FUNCTION_BLOCK Doors (* Composite Function Block Type *)
  (* Standard: 61499-2 *)
  (* Version 0.0, 11/8/2016, Dmitry, nxtControl GmbH, template *)
  PACKAGE Main;
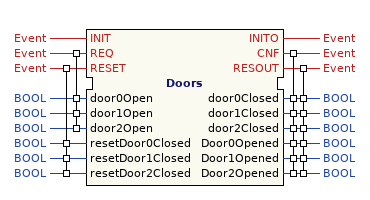
  EVENT_INPUT
    INIT; (* Initialization Request *)
    REQ WITH door0Open, door1Open, door2Open; (* Normal Execution Request *)
    RESET WITH resetDoor0Closed, resetDoor1Closed, resetDoor2Closed;
  END_EVENT
  EVENT_OUTPUT
    INITO; (* Initialization Confirm *)
    CNF WITH door0Closed, door1Closed, door2Closed, Door0Opened, Door1Opened, Door2Opened; (* Execution Confirmation *)
    RESOUT WITH door0Closed, door1Closed, door2Closed, Door0Opened, Door1Opened, Door2Opened;
  END_EVENT
  VAR_INPUT
    door0Open : BOOL;
    door1Open : BOOL;
    door2Open : BOOL;
    resetDoor0Closed : BOOL;
    resetDoor1Closed : BOOL;
    resetDoor2Closed : BOOL;
  END_VAR
  VAR_OUTPUT
    door0Closed : BOOL;
    door1Closed : BOOL;
    door2Closed : BOOL;
    Door0Opened : BOOL;
    Door1Opened : BOOL;
    Door2Opened : BOOL;
  END_VAR
  FBS
    Door0 : Door;
    Door1 : Door;
    Door2 : Door;
  END_FBS
  EVENT_CONNECTIONS
    Door0.CNF TO Door1.REQ;
    Door0.INITO TO Door1.INIT;
    Door1.CNF TO Door2.REQ;
    Door1.INITO TO Door2.INIT;
    INIT TO Door0.INIT;
    REQ TO Door0.REQ;
    Door2.INITO TO INITO;
    Door2.CNF TO CNF;
    RESET TO Door0.RESET;
    Door0.RESOUT TO Door1.RESET;
    Door1.RESOUT TO Door2.RESET;
    Door2.RESOUT TO RESOUT;
  END_CONNECTIONS
  DATA_CONNECTIONS
    door0Open TO Door0.OpenDoor;
    Door0.DoorClosed TO door0Closed;
    Door1.DoorClosed TO door1Closed;
    door1Open TO Door1.OpenDoor;
    door2Open TO Door2.OpenDoor;
    Door2.DoorClosed TO door2Closed;
    Door0.DoorOpened TO Door0Opened;
    Door1.DoorOpened TO Door1Opened;
    Door2.DoorOpened TO Door2Opened;
    resetDoor0Closed TO Door0.ResetDoorClosed;
    resetDoor1Closed TO Door1.ResetDoorClosed;
    resetDoor2Closed TO Door2.ResetDoorClosed;
  END_CONNECTIONS
END_FUNCTION_BLOCK
